FUNCTION_BLOCK InterfaceManager_test EXTENDS TcUnit.FB_TestSuite
VAR_INPUT
END_VAR
VAR_OUTPUT
END_VAR
VAR
END_VAR

test_InitTwice();

METHOD test_InitTwice
VAR_INPUT
END_VAR
VAR 
	fb_1 : InterfaceManager;
//	fb_2 : InterfaceManager;
END_VAR
TEST('test_InitTwice');



TEST_FINISHED();
END_METHOD

END_FUNCTION_BLOCK

(* stored: Version 1.1.0.1, ProductVersion 3.1.4024.6
   POU InterfaceManager_test: Id {30c1cd6d-f339-00e4-1a35-d57ebc4aab31}, SpecialFunc None
   Method test_InitTwice: Id {fb69b5fe-8ee4-0c60-166e-2e9d1eff7b35} *)
